(* IEC 61131-3 sources: automationbase/src/Equipment, 9 files *)

(* ---- EquipmentAutoStartup.st ---- *)
USING System.Timer;
NAMESPACE Simatic.Ax.AutomationBase

    {axcode:docs-v0:@simatic-ax/automationbase:StartupWarning.md}
    INTERFACE IAutoStartup
        METHOD Status : StartUpStatus
        END_METHOD
    END_INTERFACE
    // StartupTime per Equipment or per Zonemanager?
    // Decission: Each Equipment should have its own Startup.
    // Equipment knows its own startup time (it could be different between diffrent equipments)
    // and the after an error, only this equipment has execute an startup and not the whole zone which could be still in automatic
    CLASS INTERNAL EquipmentAutoStartup IMPLEMENTS IAutoStartup
        VAR PUBLIC
            StartUpTime : TIME := T#5s;
            Mode : IOperatingMode;
            Release : IRelease;
            Equipment : IEquipmentBase;
        END_VAR
        VAR PRIVATE
            _alwaysReleased : AlwaysReleasedRelease;
            _effectiveRelease : IRelease;
            _isInitialized : BOOL;
        END_VAR
        VAR PROTECTED
            ton : OnDelay;
            internalError : BOOL;
        END_VAR
        METHOD PUBLIC Status : StartUpStatus
            IF (internalError) THEN
                Status := StartUpStatus#InternalError;
                RETURN;
            END_IF;
            // Check if in Manual mode
            IF (Mode <> NULL) AND (Mode.GetOperatingMode() = OperatingModes#Manual) THEN
                Status := StartUpStatus#Manual;
                RETURN;
            END_IF;
            // Startup warning elapsed and in Automatic mode
            IF NOT(ton.output) AND ton.signal THEN
                Status := StartUpStatus#AutoStartingUp;
                RETURN;
            ELSIF (ton.output) THEN
                Status := StartUpStatus#AutoStartedUp;
                RETURN;
            ELSE
                Status := StartUpStatus#NotReleased;
                RETURN;
            END_IF;
        END_METHOD
        METHOD PUBLIC RunCyclic
            VAR_TEMP
                _runStartUpTimer : BOOL;
            END_VAR

            IF (NOT _isInitialized) THEN
                // Null-Object-Pattern: If Release is NULL, use AlwaysReleasedRelease
                IF (Release = NULL) THEN
                    _effectiveRelease := _alwaysReleased;
                ELSE
                    _effectiveRelease := Release;
                END_IF;
                _isInitialized := TRUE;
            END_IF;

            IF (mode = NULL) OR (equipment = NULL) THEN
                internalError := TRUE;
                RETURN;
            END_IF;

            _runStartUpTimer := (mode.GetOperatingMode() = OperatingModes#Automatic);
            _runStartUpTimer := _runStartUpTimer AND _effectiveRelease.IsReleased();
            _runStartUpTimer := _runStartUpTimer AND NOT(equipment.HasError());
            ton(signal := _runStartUpTimer, duration := StartUpTime);
        END_METHOD
    END_CLASS

    TYPE
        StartUpStatus : (InternalError, NotReleased, Manual, AutoStartingUp, AutoStartedUp) := NotReleased;
    END_TYPE

END_NAMESPACE

(* ---- ErrorStates.st ---- *)
USING System.Timer;

NAMESPACE Simatic.Ax.AutomationBase
    /// Error state codes for equipment
    /// NoError: No error present (0x0000)
    /// ConfigError: Configuration error, typically Mode not assigned (0x8001)
    /// OtherError: Equipment-specific error (0x8999)
    TYPE
        ErrorState : WORD (NoError := WORD#0000, ConfigError := WORD#8001, OtherError := WORD#8999) := NoError;
    END_TYPE
END_NAMESPACE

(* ---- IEquipmentBase.st ---- *)
NAMESPACE Simatic.Ax.AutomationBase

    {axcode:docs-v0:@simatic-ax/automationbase:EquipmentBase.md}
    /// Interface for equipment base functionality
    /// Defines the contract for equipment lifecycle management
    INTERFACE IEquipmentBase
        /// Main cyclic method - must be called every PLC cycle
        METHOD RunCyclic
        END_METHOD

        /// Returns TRUE if equipment has an error
        METHOD HasError : BOOL
        END_METHOD

        /// Returns the current error code
        METHOD GetError : WORD
        END_METHOD

        /// Sets an error state
        METHOD SetError
            VAR_INPUT
                errorState : WORD;
            END_VAR
        END_METHOD

        /// Sets an error state with error text
        METHOD SetError
            VAR_INPUT
                errorState : WORD;
                errorText : STRING[30];
            END_VAR
        END_METHOD

        /// Returns the last error message
        METHOD GetErrorText : STRING[30]
        END_METHOD

        /// Returns the current startup status
        METHOD GetStartupStatus : StartUpStatus
        END_METHOD

        /// Resets the fault state and clears error message
        METHOD ResetFault
        END_METHOD
    END_INTERFACE

END_NAMESPACE

(* ---- IRelease.st ---- *)
NAMESPACE Simatic.Ax.AutomationBase

    {axcode:docs-v0:@simatic-ax/automationbase:Release.md}
    /// Interface for release providers
    /// Implement this to control when equipment is allowed to start
    /// Used for safety interlocks, upstream dependencies, etc.
    INTERFACE IRelease
        /// Returns TRUE when equipment is released and allowed to operate
        METHOD IsReleased : BOOL
        END_METHOD
    END_INTERFACE

END_NAMESPACE

(* ---- IResetCommand.st ---- *)
NAMESPACE Simatic.Ax.AutomationBase

    /// Interface for reset command providers
    /// Implement this to provide centralized reset commands to equipment
    INTERFACE IResetCommand
        /// Returns TRUE when a reset command is active
        /// Equipment calls this to check if reset should be attempted
        METHOD ResetFaultRequest : BOOL
        END_METHOD

        /// Equipment calls this to report it has an active error
        /// Call this every cycle when equipment has an error
        METHOD ReportError
        END_METHOD

    END_INTERFACE

END_NAMESPACE

(* ---- AlwaysReleasedRelease.st ---- *)
NAMESPACE Simatic.Ax.AutomationBase

    /// Null-Object implementation of IRelease that always returns TRUE
    /// This is used as default when no release strategy is configured
    CLASS INTERNAL AlwaysReleasedRelease IMPLEMENTS IRelease
        METHOD PUBLIC IsReleased : BOOL
            IsReleased := TRUE;
        END_METHOD
    END_CLASS

    /// Simple release implementation that directly exposes a BOOL as release state
    CLASS BoolRelease IMPLEMENTS IRelease
        VAR PUBLIC
            ReleaseSignal : BOOL;
        END_VAR

        METHOD PUBLIC IsReleased : BOOL
            IsReleased := ReleaseSignal;
        END_METHOD
    END_CLASS

END_NAMESPACE

(* ---- BinSignalRelease.st ---- *)
USING Simatic.Ax.IO.Input;

NAMESPACE Simatic.Ax.AutomationBase

    /// Release implementation that evaluates an IBinSignal
    CLASS BinSignalRelease IMPLEMENTS IRelease
        VAR PUBLIC
            ReleaseSignal : IBinSignal;
        END_VAR

        METHOD PUBLIC IsReleased : BOOL
            IF (ReleaseSignal = NULL) THEN
                IsReleased := FALSE;
                RETURN;
            END_IF;

            IsReleased := ReleaseSignal.Q();
        END_METHOD
    END_CLASS

END_NAMESPACE

(* ---- EquipmentBase.st ---- *)
NAMESPACE Simatic.Ax.AutomationBase

    {axcode:docs-v0:@simatic-ax/automationbase:EquipmentBase.md}
    /// Abstract base class for all equipment
    /// Provides initialization, cyclic execution, error handling, and automatic startup
    /// Inherit from this class and implement InitUser() and RunCyclicUserCode()
    CLASS ABSTRACT EquipmentBase
        IMPLEMENTS IEquipmentBase
        VAR PUBLIC
            /// Duration of startup warning phase before equipment is fully started (default: 5 seconds)
            StartUpTime : TIME := T#5s;

            /// Operating mode provider (MANDATORY - must be assigned)
            Mode : IOperatingMode;

            /// External release provider (optional - if NULL, equipment is always released)
            ExternalRelease : IRelease;

            /// Custom auto-startup implementation (optional - if NULL, uses internal default)
            ExternalAutoStartup : IAutoStartup;

            /// Reset command provider (optional - if NULL, no automatic reset)
            ResetCommand : IResetCommand;
        END_VAR
        VAR PRIVATE
            /// Flag indicating if equipment has been initialized
            isInitialized : BOOL;

            /// Internal default auto-startup implementation
            _defaultAutoStartup : EquipmentAutoStartup;

            /// Active auto-startup instance (either external or default)
            _autoRelease : IAutoStartup;

            /// Flag indicating if default auto-startup is being used
            _useDefaultAutoStartup : BOOL;

            /// stores the current startup status of the equipment
            _startupStatus : StartUpStatus;
        END_VAR
        VAR PROTECTED
            /// Equipment has any error
            _hasError : BOOL;

            /// Current error state
            _errorState : WORD;

            /// Last error message
            _errorText : STRING[30];
        END_VAR

        /// Main cyclic method - call this every PLC cycle
        /// Handles automatic initialization on first call
        METHOD PUBLIC RunCyclic
            VAR_TEMP
                noConfigError : BOOL;
                resetCommandActive : BOOL;
            END_VAR
            IF NOT (isInitialized) THEN
                THIS.Init();
            END_IF;

            noConfigError := _errorState <> ErrorState#ConfigError;
            _hasError := _errorState <> ErrorState#NoError;
            IF (noConfigError) THEN
                // Only run default auto startup if no external auto startup is provided
                IF (_useDefaultAutoStartup) THEN
                    _defaultAutoStartup.RunCyclic();
                END_IF;
                THIS.RunCyclicUserCode();
            END_IF;

            // Handle automatic reset command if configured
            IF (ResetCommand <> NULL) THEN
                resetCommandActive := ResetCommand.ResetFaultRequest();
                IF (resetCommandActive AND _hasError) THEN
                    THIS.ResetFault();
                END_IF;

            // Report error status to reset manager if configured
            IF (ResetCommand <> NULL AND _hasError) THEN
                ResetCommand.ReportError();
            END_IF;

            END_IF;

        END_METHOD

        /// Private initialization method - called automatically on first RunCyclic()
        /// Configures auto-startup and validates configuration
        METHOD PRIVATE Init
            IF (ExternalAutoStartup <> NULL) THEN
                _autoRelease := ExternalAutoStartup;
                _useDefaultAutoStartup := FALSE;
            ELSE
                _defaultAutoStartup.StartUpTime := StartUpTime;
                _defaultAutoStartup.Release := ExternalRelease;
                _defaultAutoStartup.Mode := Mode;
                _defaultAutoStartup.Equipment := THIS;
                _autoRelease := _defaultAutoStartup;  // set auto release to default behavior
                _useDefaultAutoStartup := TRUE;
            END_IF;
            IF (Mode = NULL) THEN
                THIS.SetError(errorState := ErrorState#ConfigError);
            END_IF;

            THIS.InitUser();
            isInitialized := TRUE;
        END_METHOD
        /// Abstract method for cyclic user code
        /// Implement this in derived classes for equipment-specific logic
        METHOD PROTECTED ABSTRACT RunCyclicUserCode
        END_METHOD

        /// Abstract method for user initialization
        /// Implement this in derived classes for equipment-specific initialization
        METHOD PROTECTED ABSTRACT InitUser
        END_METHOD

        /// Returns TRUE if equipment has an error
        METHOD PUBLIC HasError : BOOL
            HasError := _hasError;
        END_METHOD

        /// Returns the current startup status
        METHOD PUBLIC GetStartupStatus : StartUpStatus
            IF _autoRelease = NULL THEN
                GetStartupStatus := StartUpStatus#InternalError;
                RETURN;
            END_IF;
            _startupStatus := _autoRelease.Status();
            GetStartupStatus := _startupStatus;
        END_METHOD

        /// Returns the current error code
        METHOD PUBLIC GetError : WORD
            GetError := _errorState;
        END_METHOD

        /// Sets an error state
        METHOD PUBLIC SetError
            VAR_INPUT
                errorState : WORD;
            END_VAR
            _errorState := errorState;
            _errorText := '';
        END_METHOD

        /// Sets an error state with error text
        METHOD PUBLIC SetError
            VAR_INPUT
                errorState : WORD;
                errorText : STRING[30];
            END_VAR
            _errorState := errorState;
            _errorText := errorText;
            IF (errorState <> ErrorState#NoError) THEN
                _hasError := TRUE;
            END_IF;
        END_METHOD

        /// Returns the last error message
        METHOD PUBLIC GetErrorText : STRING[30]
            GetErrorText := _errorText;
        END_METHOD

        /// Resets the fault state and clears error message
        METHOD PUBLIC ResetFault
            IF (THIS.ResetFaultUser()) THEN
                _errorState := ErrorState#NoError;
                _errorText := '';
                _hasError := FALSE;
            END_IF;
        END_METHOD

        /// User-specific reset logic (can be overridden in derived classes)
        /// Default implementation clears error state and text
        METHOD ABSTRACT ResetFaultUser : BOOL
        END_METHOD
    END_CLASS

END_NAMESPACE

(* ---- ResetCommandManager.st ---- *)
USING Simatic.Ax.IO.Input;

NAMESPACE Simatic.Ax.AutomationBase

    /// Simple and robust reset command manager
    /// Equipment reports errors via ReportError() every cycle while error is active
    /// Manager provides reset command that is active for exactly one cycle
    /// Reset is triggered on rising edge of ResetSignal
    CLASS ResetCommandManager IMPLEMENTS IResetCommand
        VAR PUBLIC
            /// Reset signal input (connect to HMI button or other signal source)
            /// Reset is triggered on rising edge via QRis()
            ResetSignal : IBinSignal;
        END_VAR

        VAR PRIVATE
            /// TRUE if any equipment has reported an error in current cycle
            _anyErrorIsActive : BOOL;

            /// TRUE if reset command is active (valid for exactly one cycle)
            _resetCommandActive : BOOL;
        END_VAR

        /// Call this every cycle to update reset command state
        /// Reset command is cleared at start and only set on rising edge of ResetSignal
        /// This ensures reset command is active for exactly one cycle
        METHOD PUBLIC RunCyclic
            // Clear reset command at start of cycle
            _resetCommandActive := FALSE;

            // Detect rising edge of reset signal and activate reset command
            IF (ResetSignal <> NULL AND ResetSignal.QRis()) THEN
                _resetCommandActive := TRUE;
                _anyErrorIsActive := FALSE; // Clear error flag on reset
            END_IF;
        END_METHOD

        /// Returns TRUE when a reset command is active
        /// Equipment calls this to check if reset should be attempted
        METHOD PUBLIC ResetFaultRequest : BOOL
            ResetFaultRequest := _resetCommandActive;
        END_METHOD

        /// Equipment calls this to report it has an active error
        /// Must be called every cycle while equipment has an error
        METHOD PUBLIC ReportError
            _anyErrorIsActive := TRUE;
        END_METHOD

        /// Returns TRUE if any equipment has reported an active error
        METHOD PUBLIC AnyErrorActive : BOOL
            AnyErrorActive := _anyErrorIsActive;
        END_METHOD

        /// Returns TRUE if reset command is currently active
        METHOD PUBLIC IsResetActive : BOOL
            IsResetActive := _resetCommandActive;
        END_METHOD
    END_CLASS

END_NAMESPACE
